{attribute 'GeneratedUsingTerminal: EL4002-0000-0018'}
{attribute addProperty BoxType "EL4002-0000-0018"}
{attribute addProperty Id "Analog_outputAT %Q*INT2"}
{attribute addProperty CRC "3128867708"}
{attribute addProperty Size "2"}
TYPE AO_Output_Channel_BA7EBB7C :
STRUCT
	{attribute addProperty Name "Analog_output"}
	Analog_output AT %Q* : INT;
END_STRUCT
END_TYPE

(* stored: Version 1.2.0.0, ProductVersion 3.1.4024.9
   DUT AO_Output_Channel_BA7EBB7C: Id {6b5b9220-1131-4e10-8d61-67f02a7b7562} *)
